// TIA Portal V18 export
DATA_BLOCK "Drill_DB"   // DB30
// stored: AutoNumber false, InstanceOfName Drill, InstanceOfType FB
"Drill"
   // VAR_INPUT
   //    DrillPSISet : Real;
   //    DisableThrottle : Bool;
   // END_VAR
   // VAR_OUTPUT
   //    FlowFwdmAOut : Real;
   //    FwdEnableP1 : Bool;
   //    TorquePSIOut : Real;
   //    FwdEnableP2 : Bool;
   // END_VAR
   // VAR
   //    PSinitialize : Bool;
   //    TorqLowLimitFtLbs { ExternalAccessible := 'False'; ExternalVisible := 'False'; ExternalWritable := 'False'} : Real;
   //    TorqHighLimitFtLbs : Real;
   //    TorqLimiting : Bool;
   //    TorqLimitTrig : Bool;
   //    LimitFlowmAOut : Real;
   //    TorqLimit_TON { S7_SetPoint := 'True'} : TON_TIME;
   //    TorqLimit_SlewDec { S7_SetPoint := 'True'} : "SlewDec";
   //    Torq_Limit_SlewInc { S7_SetPoint := 'True'} : "SlewInc";
   // END_VAR
BEGIN
END_DATA_BLOCK
